(* IEC 61131-3 sources: stopGate_FuB/Logical/Libraries/runtime, 3 files *)

(* ---- runtime.typ ---- *)
TYPE
	SFCActionType : STRUCT			(*internal use*)
		x	: BOOL;
		_x	: BOOL;
		t	: TIME;
		_t	: TIME;
		AC	: SFCActionControl;
	END_STRUCT;
	SFCActionType2 : STRUCT		(*internal use*)
		x	: BOOL;
		_x	: BOOL;
		AC	: SFCAC2;
	END_STRUCT;
	SFCActionCType : STRUCT		(*internal use*)
		x		: BOOL;
		_x		: BOOL;
		force	: BOOL;
		_force	: BOOL;
		active	: BOOL;
		_active	: BOOL;
		error	: BOOL;
		AC		: SFCActionControl;
	END_STRUCT;
	SFCActionCType2 : STRUCT	(*internal use*)
		x		: BOOL;
		_x		: BOOL;
		force	: BOOL;
		_force	: BOOL;
		active	: BOOL;
		_active	: BOOL;
		error	: BOOL;
		AC		: SFCAC2;
	END_STRUCT;
	SFCActionCType3 : STRUCT	(*internal use*)
		t		: LREAL;
		_t		: LREAL;
		tp		: LREAL;
		x		: BOOL;
		_x		: BOOL;
		force	: BOOL;
		_force	: BOOL;
		active	: BOOL;
		_active	: BOOL;
		error	: BOOL;
		AC		: SFCAC3;
	END_STRUCT;
	SFCStepType : STRUCT			(*internal use*)
		x	: BOOL;
		t	: TIME;
		_x	: BOOL;
		_t	: TIME;
	END_STRUCT;
	SFCStepCType : STRUCT		(*internal use*)
		t					: TIME;
		_t					: TIME;
		inactive_actions	: UDINT;
		_inactive_actions	: UDINT;
		error_actions		: UDINT;
		x					: BOOL;
		_x					: BOOL;
		x_activate			: BOOL;
		force				: BOOL;
		_force				: BOOL;
		active				: BOOL;
		_active				: BOOL;
		error				: BOOL;
		tip					: BOOL;
		tip_disable_duration: BOOL;
		tip_disable_action	: BOOL;
	END_STRUCT;
	SFCStepCType3 : STRUCT		(*internal use*)
		t						: LREAL;
		_t						: LREAL;
		tp						: LREAL;
		inactive_actions		: UDINT;
		_inactive_actions		: UDINT;
		error_actions			: UDINT;
		x						: BOOL;
		_x						: BOOL;
		x_activate				: {REDUND_UNREPLICABLE} BOOL;
		force					: BOOL;
		_force					: BOOL;
		active					: BOOL;
		_active					: BOOL;
		error					: BOOL;
		tip						: BOOL;
		tip_disable_duration	: BOOL;
		tip_disable_action		: BOOL;
	END_STRUCT;
	SFCSimpleStepCType : STRUCT	(*internal use*)
		t						: TIME;
		_t						: TIME;
		x						: BOOL;
		_x						: BOOL;
		x_activate				: BOOL;
		force					: BOOL;
		_force					: BOOL;
		active					: BOOL;
		_active					: BOOL;
		error					: BOOL;
		tip						: BOOL;
		tip_disable_duration	: BOOL;
		tip_disable_action		: BOOL;
	END_STRUCT;
	SFCSimpleStepCType3 : STRUCT	(*internal use*)
		t						: LREAL;
		_t						: LREAL;
		tp						: LREAL;
		x						: BOOL;
		_x						: BOOL;
		x_activate				: {REDUND_UNREPLICABLE} BOOL;
		force					: BOOL;
		_force					: BOOL;
		active					:  BOOL;
		_active					: BOOL;
		error					: BOOL;
		tip						: BOOL;
		tip_disable_duration	: BOOL;
		tip_disable_action		: BOOL;
	END_STRUCT;
	SFCTransitionCType : STRUCT	(*internal use*)
		force	: BOOL;
		_force	: BOOL;
		active	: BOOL;
		_active	: BOOL;
	END_STRUCT;
	TimerType : STRUCT	(*internal use*)
		ptime	: LREAL;
		etime	: LREAL;
		start	: LREAL;
		in		: USINT;
		q		: USINT;
	END_STRUCT;

	ArFBStateInternalType : STRUCT			(*fb state machine internal context*)
		ExecuteRef		: UDINT;
		BusyRef			: UDINT;
		DoneRef			: UDINT;
		ErrorRef		: UDINT;
		ActiveRef		: UDINT;
		StatusRef		: UDINT;
		FBCyclic		: UDINT;
		AsyfumaState		: UDINT;
		FBResetOut		: UDINT;
		Argument		: UDINT;
		State			: UDINT;
		ExecutePrev		: BOOL;
	END_STRUCT;

	ArFBAsyFuMaInternalType : STRUCT		(*asynchronous function manager internal context*)
		State			: UINT;
		Result			: DINT;
	END_STRUCT;

END_TYPE

(* ---- runtime.fun ---- *)
{REDUND_OK} FUNCTION_BLOCK r_trig 			(*for internal use only - do not use this function in user programs*)
	VAR_INPUT
		CLK	:BOOL;
	END_VAR
	VAR_OUTPUT
		Q	:BOOL;
	END_VAR
	VAR
		M	:BOOL;
	END_VAR
END_FUNCTION_BLOCK
{REDUND_OK} FUNCTION_BLOCK f_trig 			(*for internal use only - do not use this function in user programs*)
	VAR_INPUT
		CLK	:BOOL;
	END_VAR
	VAR_OUTPUT
		Q	:BOOL;
	END_VAR
	VAR
		M	:BOOL;
	END_VAR
END_FUNCTION_BLOCK
{REDUND_OK} FUNCTION_BLOCK rf_trig 			(*for internal use only - do not use this function in user programs*)
	VAR_INPUT
		CLK	:BOOL;
	END_VAR
	VAR_OUTPUT
		Q	:BOOL;
	END_VAR
	VAR
		M	:BOOL;
	END_VAR
END_FUNCTION_BLOCK
FUNCTION GetTime : TIME 		(*for internal use only - do not use this function in user programs*)
END_FUNCTION
{REDUND_OK} FUNCTION_BLOCK SFCActionControl (*for internal use only - do not use this function in user programs*)
	VAR_INPUT
		N	:BOOL;
		R0	:BOOL;
		S0	:BOOL;
		L	:BOOL;
		D	:BOOL;
		P	:BOOL;
		SD	:BOOL;
		DS	:BOOL;
		SL	:BOOL;
		T	:TIME;
	END_VAR
	VAR_OUTPUT
		Q	:BOOL;
	END_VAR
	VAR
		S_FF_SET	:USINT;
		S_FF_R1		:USINT;
		S_FF_Q		:USINT;
		dummy1		:USINT;
		L_TMR_PT	:TIME;
		L_TMR_ET	:TIME;
		L_TMR_STAR	:TIME;
		L_TMR_IN	:USINT;
		L_TMR_Q		:USINT;
		L_TMR_M		:USINT;
		dummy2		:USINT;
		D_TMR_PT	:TIME;
		D_TMR_ET	:TIME;
		D_TMR_STAR	:TIME;
		D_TMR_IN	:USINT;
		D_TMR_Q		:USINT;
		D_TMR_M		:USINT;
		dummy3		:USINT;
		P_TRIG_CLK	:USINT;
		P_TRIG_Q	:USINT;
		P_TRIG_M	:USINT;
		dummy4		:USINT;
		SD_TMR_PT	:TIME;
		SD_TMR_ET	:TIME;
		SD_TMR_STA	:TIME;
		SD_TMR_IN	:USINT;
		SD_TMR_Q	:USINT;
		SD_TMR_M	:USINT;
		dummy5		:USINT;
		SD_FF_SET	:USINT;
		SD_FF_R1	:USINT;
		SD_FF_Q		:USINT;
		DS_FF_SET	:USINT;
		DS_FF_R1	:USINT;
		DS_FF_Q		:USINT;
		DS_TMR_PT	:TIME;
		DS_TMR_ET	:TIME;
		DS_TMR_STA	:TIME;
		DS_TMR_IN	:USINT;
		DS_TMR_Q	:USINT;
		DS_TMR_M	:USINT;
		dummy6		:USINT;
		SL_FF_SET	:USINT;
		SL_FF_R1	:USINT;
		SL_FF_Q		:USINT;
		dummy7		:USINT;
		SL_TMR_PT	:TIME;
		SL_TMR_ET	:TIME;
		SL_TMR_STA	:TIME;
		SL_TMR_IN	:USINT;
		SL_TMR_Q	:USINT;
		SL_TMR_M	:USINT;
		dummy8		:USINT;
	END_VAR
END_FUNCTION_BLOCK
{REDUND_OK} FUNCTION_BLOCK SFCAC2				(*for internal use only - do not use this function in user programs*)
	VAR_INPUT
		N	: {REDUND_UNREPLICABLE} BOOL;
		R0	: {REDUND_UNREPLICABLE} BOOL;
		S0	: {REDUND_UNREPLICABLE} BOOL;
		L	: {REDUND_UNREPLICABLE} BOOL;
		D	: {REDUND_UNREPLICABLE} BOOL;
		P	: {REDUND_UNREPLICABLE} BOOL;
		P1	: {REDUND_UNREPLICABLE} BOOL;
		P0	: {REDUND_UNREPLICABLE} BOOL;
		SD	: {REDUND_UNREPLICABLE} BOOL;
		DS	: {REDUND_UNREPLICABLE} BOOL;
		SL	: {REDUND_UNREPLICABLE} BOOL;
		T	:TIME;
	END_VAR
	VAR_OUTPUT
		Q	:BOOL;
		A	:BOOL;
	END_VAR
	VAR
		S_FF_SET	:USINT;
		S_FF_R1		:USINT;
		S_FF_Q		:USINT;
		L_TMR_PT	:TIME;
		L_TMR_ET	:TIME;
		L_TMR_STAR	:TIME;
		L_TMR_IN	:USINT;
		L_TMR_Q		:USINT;
		L_TMR_M		:USINT;
		D_TMR_PT	:TIME;
		D_TMR_ET	:TIME;
		D_TMR_STAR	:TIME;
		D_TMR_IN	:USINT;
		D_TMR_Q		:USINT;
		D_TMR_M		:USINT;
		SD_TMR_PT	:TIME;
		SD_TMR_ET	:TIME;
		SD_TMR_STA	:TIME;
		SD_TMR_IN	:USINT;
		SD_TMR_Q	:USINT;
		SD_TMR_M	:USINT;
		SD_FF_SET	:USINT;
		SD_FF_R1	:USINT;
		SD_FF_Q1	:USINT;
		DS_FF_SET	:USINT;
		DS_FF_R1	:USINT;
		DS_FF_Q1	:USINT;
		DS_TMR_PT	:TIME;
		DS_TMR_ET	:TIME;
		DS_TMR_STA	:TIME;
		DS_TMR_IN	:USINT;
		DS_TMR_Q	:USINT;
		DS_TMR_M	:USINT;
		SL_FF_SET	:USINT;
		SL_FF_R1	:USINT;
		SL_FF_Q		:USINT;
		SL_TMR_PT	:TIME;
		SL_TMR_ET	:TIME;
		SL_TMR_STA	:TIME;
		SL_TMR_IN	:USINT;
		SL_TMR_Q	:USINT;
		SL_TMR_M	:USINT;
		P_TRIG_Q	:USINT;
		P_TRIG_M	:USINT;
		Q_TRIG_Q	:USINT;
		Q_TRIG_M	:USINT;
		P1_TRIG_Q	:USINT;
		P1_TRIG_M	:USINT;
		P0_TRIG_Q	:USINT;
		P0_TRIG_M	:USINT;
	END_VAR
END_FUNCTION_BLOCK
{REDUND_OK} FUNCTION RealTan : LREAL
	VAR_INPUT
		x	:LREAL;
	END_VAR
END_FUNCTION
{REDUND_OK} FUNCTION RealAtan : LREAL
	VAR_INPUT
		x	:LREAL;
	END_VAR
END_FUNCTION
{REDUND_OK} FUNCTION RealAsin : LREAL
	VAR_INPUT
		x	:LREAL;
	END_VAR
END_FUNCTION
{REDUND_OK} FUNCTION RealAcos : LREAL
	VAR_INPUT
		x	:LREAL;
	END_VAR
END_FUNCTION
{REDUND_OK} FUNCTION RealExp : LREAL
	VAR_INPUT
		x	:LREAL;
	END_VAR
END_FUNCTION
{REDUND_OK} FUNCTION RealLn : LREAL
	VAR_INPUT
		x	:LREAL;
	END_VAR
END_FUNCTION
{REDUND_OK} FUNCTION RealLog : LREAL
	VAR_INPUT
		x	:LREAL;
	END_VAR
END_FUNCTION
{REDUND_OK} FUNCTION RealExpt : LREAL
	VAR_INPUT
		x	:LREAL;
		y	:LREAL;
	END_VAR
END_FUNCTION
{REDUND_OK} FUNCTION RealAbs : LREAL
	VAR_INPUT
		x	:LREAL;
	END_VAR
END_FUNCTION
{REDUND_OK} FUNCTION RealSin : LREAL
	VAR_INPUT
		x	:LREAL;
	END_VAR
END_FUNCTION
{REDUND_OK} FUNCTION RealCos : LREAL
	VAR_INPUT
		x	:LREAL;
	END_VAR
END_FUNCTION
{REDUND_OK} FUNCTION RealSqrt : LREAL
	VAR_INPUT
		x	:LREAL;
	END_VAR
END_FUNCTION
{REDUND_OK} FUNCTION_BLOCK SFCAC3				(*for internal use only - do not use this function in user programs*)
	VAR_INPUT
		N		: {REDUND_UNREPLICABLE} BOOL;
		R0		: {REDUND_UNREPLICABLE} BOOL;
		S0		: {REDUND_UNREPLICABLE} BOOL;
		L		: {REDUND_UNREPLICABLE} BOOL;
		D		: {REDUND_UNREPLICABLE} BOOL;
		P		: {REDUND_UNREPLICABLE} BOOL;
		P1		: {REDUND_UNREPLICABLE} BOOL;
		P0		: {REDUND_UNREPLICABLE} BOOL;
		SD		: {REDUND_UNREPLICABLE} BOOL;
		DS		: {REDUND_UNREPLICABLE} BOOL;
		SL		: {REDUND_UNREPLICABLE} BOOL;
		T		:LREAL;
		T_ACT	: {REDUND_UNREPLICABLE} LREAL;
		PAUSE	: {REDUND_UNREPLICABLE} BOOL;
	END_VAR
	VAR_OUTPUT
		Q	: {REDUND_UNREPLICABLE} BOOL;
		A	:BOOL;
	END_VAR
	VAR
		L_TMR		:TimerType;
		D_TMR		:TimerType;
		SD_TMR		:TimerType;
		DS_TMR		:TimerType;
		SL_TMR		:TimerType;
		S_FF_Q1		:USINT;
		SD_FF_Q1	:USINT;
		DS_FF_Q1	:USINT;
		SL_FF_Q1	:USINT;
		P_R_TRIG_Q	: {REDUND_UNREPLICABLE} USINT;
		P_R_TRIG_M	:USINT;
		Q_F_TRIG_Q	: {REDUND_UNREPLICABLE} USINT;
		Q_F_TRIG_M	:USINT;
		P1_R_TRIG_Q	: {REDUND_UNREPLICABLE} USINT;
		P1_R_TRIG_M	:USINT;
		P0_F_TRIG_Q	: {REDUND_UNREPLICABLE} USINT;
		P0_F_TRIG_M	:USINT;
	END_VAR
END_FUNCTION_BLOCK

(* ---- runtime.var ---- *)
 (*Common Functionblock Status*)
VAR CONSTANT
	ERR_OK                : UINT := 0;			(*no error*)
	ERR_NOTIMPLEMENTED    : UINT := 9999;       (*function or function block not implemented*)
	ERR_FUB_ENABLE_FALSE  : UINT := 16#FFFE;	(*function block parameter "enable" is FALSE*)
	ERR_FUB_BUSY          : UINT := 16#FFFF;	(*function block still working*)
	ERR_FUB_REDUNDANT     :	UINT := 35688;		(*This FUB can not be used on the standby CPU*)
	ERR_FB_NOT_IMPLEMENTED: DINT := -1070585592;(*function or function block not implemented for the target system*)
END_VAR

(*IEC 61131-3 Datatypes*)
VAR CONSTANT
	IEC_DATATYPE_BOOL		: UINT := 1;		(*8 Bit containing a boolean value FALSE=0 or TRUE=1*)
	IEC_DATATYPE_SINT		: UINT := 2;		(*8 Bit signed integer*)
	IEC_DATATYPE_INT		: UINT := 3;		(*16 Bit signed integer*)
	IEC_DATATYPE_DINT		: UINT := 4;		(*32 Bit signed integer*)
	IEC_DATATYPE_USINT		: UINT := 5;		(*8 Bit unsigned integer*)
	IEC_DATATYPE_UINT		: UINT := 6;		(*16 Bit unsigned integer*)
	IEC_DATATYPE_UDINT		: UINT := 7;		(*32 Bit unsigned integer*)
	IEC_DATATYPE_REAL		: UINT := 8;		(*32 Bit floating point number*)
	IEC_DATATYPE_STRING		: UINT := 9;		(*Variable-length single-byte character string*)
	IEC_DATATYPE_ULINT		: UINT := 10;		(*64 Bit unsigned integer*)
	IEC_DATATYPE_DATE_AND_TIME	: UINT := 11;	(*32 Bit of Date in Seconds since 01.01.1970 00:00:00*)
	IEC_DATATYPE_TIME		: UINT := 12;		(*32 Bit of Time in ms*)
	IEC_DATATYPE_DATE		: UINT := 13;		(*32 Bit of Date (only)*)
	IEC_DATATYPE_LREAL		: UINT := 14;		(*64 Bit floating point number*)
	IEC_DATATYPE_TIME_OF_DAY: UINT := 16;		(*32 Bit Time of day (only)*)
	IEC_DATATYPE_BYTE		: UINT := 17;		(*Bit string of length 8*)
	IEC_DATATYPE_WORD		: UINT := 18;		(*Bit string of length 16*)
	IEC_DATATYPE_DWORD		: UINT := 19;		(*Bit string of length 32*)
	IEC_DATATYPE_LWORD		: UINT := 20;		(*Bit string of length 64*)
	IEC_DATATYPE_WSTRING	: UINT := 21;		(*Variable-length double-byte character string*)
	IEC_DATATYPE_LINT		: UINT := 23;		(*64 Bit signed integer*)
END_VAR
